PROGRAM P_LocalTest
VAR
	fbLocalTest : FB_LocalTest;
END_VAR

fbLocalTest(
	fTime := G_OPC.fTime,
	bEnableTest := G_Enables.bLocalTest,
	
	fSignal => G_OPC.fValveOneOutput
);

END_PROGRAM

(* stored: Version 1.1.0.1
   POU P_LocalTest: Id {fcefc10f-7bcc-4bcc-b662-2324f5ab3460}, SpecialFunc None *)
